// TwinCAT 3 PLC project PLC
// ProgramVersion: 3.1.4026.9
// libraries:
//   Tc2_MC2, * (Beckhoff Automation GmbH)
//   Tc2_Standard, * (Beckhoff Automation GmbH)
//   Tc2_System, * (Beckhoff Automation GmbH)
// project tree:
//   DUTs/ MoveState_t.TcDUT
//   GVLs/ GVL.TcGVL
//   / PlcTask.TcTTO
//   POUs/ FB_Cylinder.TcPOU, MAIN.TcPOU, Motion.TcPOU
// real-time tasks:
//   TASK PlcTask: cycle T#10ms, priority 20, ADS port 350
// motion (NC):
//   TASK NC-Task 1 SAF: cycle T#2ms, priority 4, ADS port 501
//   TASK NC-Task 1 SVB: cycle T#10ms, priority 8, ADS port 511
//   AXIS Axis 1 (id 1)
//     OtherSettings: AllowMotionCmdToSlave=true
//     encoder EncType=1
//     drive DrvType=5
//       Analog: TorqueSetpointScale=10, ScaleFactorActTorque=0.1
//       TimeComp: TaskDelayCycles=1
//     controller CtrType=1
//       CtrPara: PriorControlFactor=1
//         Observer: BandWidth=20
// variable links:
//   PLC/PLC Instance <-> NC-Task 1 SAF/Axes/Axis 1
//     PlcTask Inputs/Motion.Axis1.NcToPlc <-> Outputs/ToPlc
//     PlcTask Outputs/Motion.Axis1.PlcToNc <-> Inputs/FromPlc

CONFIGURATION PLC
    RESOURCE PLC ON TwinCAT3
        TASK PlcTask(INTERVAL := T#10ms, PRIORITY := 20);
        PROGRAM MAIN WITH PlcTask : MAIN;
    END_RESOURCE
END_CONFIGURATION

// ---- DUTs/MoveState_t.TcDUT
TYPE MoveState_t :
(
	MOVESTATE_INIT,
	MOVESTATE_ENABLE,
	MOVESTATE_FORWARD,
	MOVESTATE_BACKWARDS,
	MOVESTATE_BACKWARDSSLOW,
	MOVESTATE_NEWTARGETPOSITION,
	MOVESTATE_ERROR,
	MOVESTATE_RESET
) UDINT;
END_TYPE

// ---- GVLs/GVL.TcGVL
{attribute 'qualified_only'}
VAR_GLOBAL
	bAuto		: BOOL;
	bRunning	: BOOL;
END_VAR

// ---- POUs/MAIN.TcPOU
PROGRAM MAIN
VAR
	Cylinders		: ARRAY[0..4] OF FB_Cylinder;
	i				: DINT;
	
	bAutoCmd		: BOOL;
	bManCmd			: BOOL;
	bStartCmd		: BOOL;
	bStopCmd		: BOOL;
	
	nRunTime		: REAL;
	nStopTime		: REAL;
	
	bInit			: BOOL := TRUE;
END_VAR

// added a comment!
IF bInit THEN
	Cylinders[0].Name := 'Infeed';
	Cylinders[1].Name := 'Clamp';
	Cylinders[2].Name := 'Outfeed';
	Cylinders[3].Name := 'Reject';
	Cylinders[4].Name := 'Spare';
	bInit := FALSE;
END_IF

IF NOT GVL.bAuto THEN
	FOR i := 0 TO 4 DO
		Cylinders[i].Manual();
	END_FOR
ELSE
	IF GVL.bRunning THEN
		Sim();
	END_IF
END_IF

Mode();

IF GVL.bAuto THEN
	IF GVL.bRunning THEN
		nRunTime := nRunTime + 0.02;
	ELSE
		nStopTime := nStopTime + 0.01;
	END_IF
END_IF

Motion();

ACTION Mode:
IF bAutoCmd THEN
	GVL.bAuto := TRUE;
END_IF

IF bManCmd THEN
	GVL.bAuto := FALSE;
	GVL.bRunning := FALSE;
END_IF

IF GVL.bAuto AND bStartCmd THEN
	GVL.bRunning := TRUE;
END_IF

IF GVL.bAuto AND bStopCmd THEN
	GVL.bRunning := FALSE;
END_IF
END_ACTION

METHOD Sim
VAR_INPUT
END_VAR
VAR_INST
	rand		: ARRAY[0..4] OF DRAND;
	j			: DINT;
	tonP		: TON;
END_VAR
rand[0](Seed:=TO_INT(i));
j := TO_DINT(rand[0].Num * 100);
IF j >= 0 AND j <= 4 THEN
	Cylinders[j].Extended := NOT Cylinders[j].Extended;
END_IF
END_METHOD

END_PROGRAM

// ---- POUs/FB_Cylinder.TcPOU
FUNCTION_BLOCK FB_Cylinder
VAR_INPUT
END_VAR
VAR_OUTPUT
END_VAR
VAR
	bExtended		: BOOL;
	bExtendCmd		: BOOL;
	bRetractCmd		: BOOL;
	
	sName			: STRING;
	ton				: TON;
	nState			: DINT;
END_VAR

PROPERTY Extended : BOOL
GET
Extended := bExtended;
END_GET
SET
bExtended := Extended;
END_SET
END_PROPERTY

METHOD Manual : BOOL
VAR_INPUT
END_VAR
CASE nState OF
	0:
		bExtended := FALSE;
		IF bExtendCmd THEN
			ton(IN:=TRUE, PT:=T#1S);
			IF ton.Q THEN
				nState := 1;
			END_IF
		END_IF
	1:
		bExtended := TRUE;
		IF bRetractCmd THEN
			ton(IN:=FALSE);
			nState := 0;
		END_IF
END_CASE
END_METHOD

PROPERTY Name : STRING
GET
Name := sName;
END_GET
SET
sName := Name;
END_SET
END_PROPERTY

END_FUNCTION_BLOCK

// ---- POUs/Motion.TcPOU
PROGRAM Motion
VAR
	/// axis reference data structure 
	Axis1: AXIS_REF;
	/// state machine state 
	state: MoveState_t;
	PowerAxis1: MC_Power;
	/// debug function block output data 
	PowerAxis1Out: ST_McOutputs;
	MoveAxis1: MC_MoveAbsolute;
	/// debug function block output data 
	MoveAbsoluteOut1: ST_McOutputs;
	MoveAxis2: MC_MoveAbsolute;
	/// debug function block output data 
	MoveAbsoluteOut2: ST_McOutputs;
	Reset: MC_Reset;
	/// debug function block output data 
	ResetOut: ST_McOutputs;
	
	autoOut		: F_TRIG;
END_VAR

(* update the axis status at the beginning of each cycle *)
Axis1();

autoOut(CLK:=GVL.bRunning);
IF autoOut.Q THEN
	state := MOVESTATE_RESET;
END_IF

(* move axis using a state machine *)
CASE state OF

	MOVESTATE_INIT :	(* initialisation *)
		(* initialize all function blocks *)
		MoveAxis1.Execute := FALSE;
		MoveAxis2.Execute := FALSE;
		Reset.Execute := FALSE;
		state := MOVESTATE_ENABLE;

	MOVESTATE_ENABLE :
		PowerAxis1.Enable := TRUE;
		PowerAxis1.Enable_Positive := TRUE;
		PowerAxis1.Enable_Negative := TRUE;
		IF PowerAxis1.Status THEN
			IF GVL.bRunning THEN
				state := MOVESTATE_FORWARD;
			END_IF
		ELSIF PowerAxis1.Error THEN
			state := MOVESTATE_ERROR;
		END_IF

	MOVESTATE_FORWARD :		(* start to first position *)
		MoveAxis1.Position := 1500;		(* start to intermediate tartet position *)
		MoveAxis1.Velocity := 500;		(* medium velocity level *)
		MoveAxis1.BufferMode := MC_Buffered;
		MoveAxis1.Execute := TRUE;
		IF MoveAxis1.Active  THEN
			(* axis is executing job but is not yet finished *)
			MoveAxis1.Execute := FALSE;
			(* leave this state and buffer a second command *)
			state := MOVESTATE_NEWTARGETPOSITION;
		ELSIF MoveAxis1.CommandAborted OR MoveAxis1.Error THEN
			state := MOVESTATE_ERROR;
		END_IF

	MOVESTATE_NEWTARGETPOSITION :		(* change target position while moving *)
		(* start a buffered motion command while axis is moving *)
		MoveAxis2.Position := 5000;		(* start to final target *)
		MoveAxis2.Velocity := 1500;		(* increase velocity *)
		MoveAxis2.BufferMode := MC_BlendingPrevious; 	(* use velocity of previous command till intermediate target position position *)
		MoveAxis2.Execute := TRUE;
		IF MoveAxis2.Done THEN
			MoveAxis2.Execute := FALSE;
			state := MOVESTATE_BACKWARDS;
		ELSIF MoveAxis2.CommandAborted OR MoveAxis2.Error THEN
			state := MOVESTATE_ERROR;
		END_IF

	MOVESTATE_BACKWARDS :	(* move back to initial position *)
		MoveAxis1.Position := 100;		(* position close to initial position *)
		MoveAxis1.Velocity := 2000;		(* high velocity *)
		MoveAxis1.BufferMode := MC_Buffered;
		MoveAxis1.Execute := TRUE;
		IF MoveAxis1.Active THEN
			(* axis is executing job but is not yet finished *)
			MoveAxis1.Execute := FALSE;
			(* leave this state and buffer a second command *)
			state := MOVESTATE_BACKWARDSSLOW;
		ELSIF MoveAxis1.CommandAborted OR MoveAxis1.Error THEN
			state := MOVESTATE_ERROR;
		END_IF

	MOVESTATE_BACKWARDSSLOW :	(* move back to initial position *)
		(* start a buffered motion command while axis is moving *)
		MoveAxis2.Position := 0;	(* back to initial position *)
		MoveAxis2.Velocity := 100; 	(* slow velocity *)
		MoveAxis2.BufferMode := MC_BlendingNext; 	(* use velocity from first target position *)
		MoveAxis2.Execute := TRUE;
		IF MoveAxis2.Done THEN
			MoveAxis2.Execute := FALSE;
			state := MOVESTATE_FORWARD;
		ELSIF MoveAxis2.CommandAborted OR MoveAxis2.Error THEN
			state := MOVESTATE_ERROR;
		END_IF

	MOVESTATE_ERROR :
		IF Axis1.Status.Error THEN
			state := MOVESTATE_RESET;	(* axis error requires reset *)
		ELSE
			state := MOVESTATE_INIT;		(* function block errors don't need a reset *)
		END_IF

	MOVESTATE_RESET :
		Reset.Execute := TRUE;
		IF Reset.Done THEN
			state := MOVESTATE_INIT;
		ELSIF Reset.Error THEN
			state := MOVESTATE_INIT; (* can't do anything here *)
		END_IF

END_CASE

ActPower();	(* call the power function block *)
ActMove();	(* call the move function block *)
ActReset();	(* call the reset function block *)

ACTION ActMove:
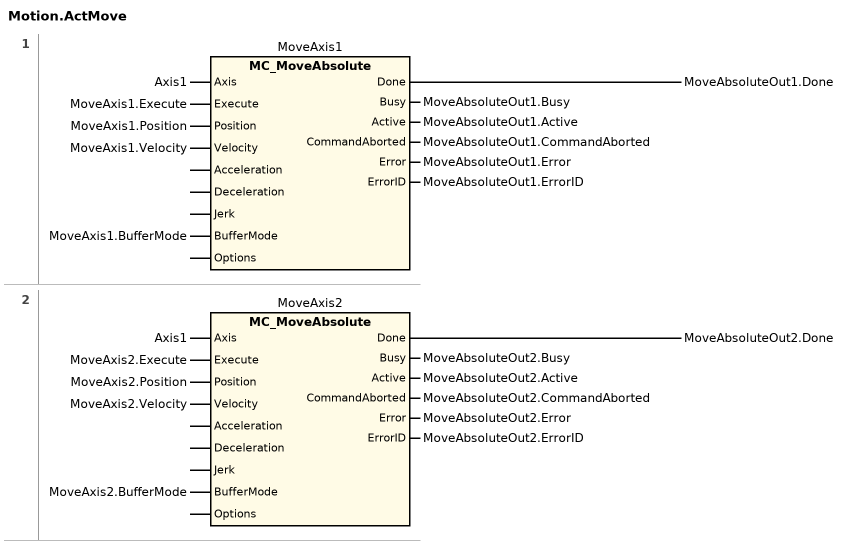
// NETWORK 1
MoveAxis1(
    Axis := Axis1,
    Execute := MoveAxis1.Execute,
    Position := MoveAxis1.Position,
    Velocity := MoveAxis1.Velocity,
    BufferMode := MoveAxis1.BufferMode,
    Busy => MoveAbsoluteOut1.Busy,
    Active => MoveAbsoluteOut1.Active,
    CommandAborted => MoveAbsoluteOut1.CommandAborted,
    Error => MoveAbsoluteOut1.Error,
    ErrorID => MoveAbsoluteOut1.ErrorID); // MC_MoveAbsolute
MoveAbsoluteOut1.Done := MoveAxis1.Done;

// NETWORK 2
MoveAxis2(
    Axis := Axis1,
    Execute := MoveAxis2.Execute,
    Position := MoveAxis2.Position,
    Velocity := MoveAxis2.Velocity,
    BufferMode := MoveAxis2.BufferMode,
    Busy => MoveAbsoluteOut2.Busy,
    Active => MoveAbsoluteOut2.Active,
    CommandAborted => MoveAbsoluteOut2.CommandAborted,
    Error => MoveAbsoluteOut2.Error,
    ErrorID => MoveAbsoluteOut2.ErrorID); // MC_MoveAbsolute
MoveAbsoluteOut2.Done := MoveAxis2.Done;
END_ACTION

ACTION ActPower:
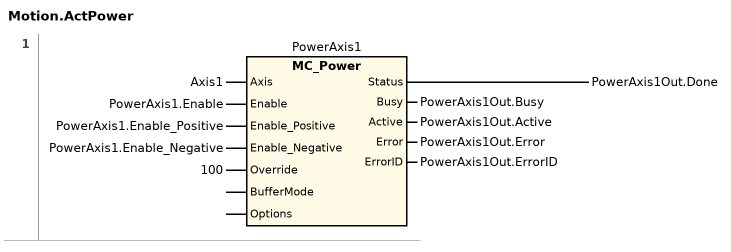
// NETWORK 1
PowerAxis1(
    Axis := Axis1,
    Enable := PowerAxis1.Enable,
    Enable_Positive := PowerAxis1.Enable_Positive,
    Enable_Negative := PowerAxis1.Enable_Negative,
    Override := 100,
    Busy => PowerAxis1Out.Busy,
    Active => PowerAxis1Out.Active,
    Error => PowerAxis1Out.Error,
    ErrorID => PowerAxis1Out.ErrorID); // MC_Power
PowerAxis1Out.Done := PowerAxis1.Status;
END_ACTION

ACTION ActReset:
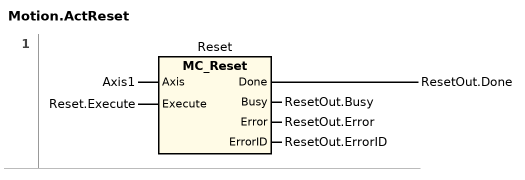
// NETWORK 1
Reset(
    Axis := Axis1,
    Execute := Reset.Execute,
    Busy => ResetOut.Busy,
    Error => ResetOut.Error,
    ErrorID => ResetOut.ErrorID); // MC_Reset
ResetOut.Done := Reset.Done;
END_ACTION

END_PROGRAM
